// TIA Portal V19 export
TYPE "C301_VAR_IF_VEN_TYPIC"
   STRUCT
      STS_AAN { ExternalAccessible := 'False'; ExternalVisible := 'False'; ExternalWritable := 'False'} : Bool;   // TRUE = Ventilator is aangestuurd FALSE = Uit
      DIR_POS { ExternalAccessible := 'False'; ExternalVisible := 'False'; ExternalWritable := 'False'} : Bool;   // TRUE = Ventilator draait in positieve richting (rijrichting)
      DIR_NEG { ExternalAccessible := 'False'; ExternalVisible := 'False'; ExternalWritable := 'False'} : Bool;   // TRUE = Ventilator draait in negatieve richting (tegenrij)
      BMO_HAND { ExternalAccessible := 'False'; ExternalVisible := 'False'; ExternalWritable := 'False'} : Bool;   // TRUE = Ventilator in hand geschakeld FALSE = niet in hand
      TYD_TOT_AAN { ExternalAccessible := 'False'; ExternalVisible := 'False'; ExternalWritable := 'False'} : LInt;   // Totaal aantal draaiuren
      TYD_TOT_AAN_UUR { ExternalAccessible := 'False'; ExternalVisible := 'False'; ExternalWritable := 'False'} : LInt;   // Totaal aantal draaiuren
      ENE_MWA1 { ExternalAccessible := 'False'; ExternalVisible := 'False'; ExternalWritable := 'False'} : Real;   // Stroommeting fase 1
      ENE_MWA2 { ExternalAccessible := 'False'; ExternalVisible := 'False'; ExternalWritable := 'False'} : Real;   // Stroommeting fase 2
      ENE_MWA3 { ExternalAccessible := 'False'; ExternalVisible := 'False'; ExternalWritable := 'False'} : Real;   // Stroommeting fase 3
      TRL_MWA { ExternalAccessible := 'False'; ExternalVisible := 'False'; ExternalWritable := 'False'} : Real;   // Trillingsmeting
      EXT_AUT { ExternalAccessible := 'False'; ExternalVisible := 'False'; ExternalWritable := 'False'} : Bool;   // Externe (hoofd) beveiliging aangesproken
      EXT_HW { ExternalAccessible := 'False'; ExternalVisible := 'False'; ExternalWritable := 'False'} : Bool;   // Sturings hardware (PLC) in storing
      STO { ExternalAccessible := 'False'; ExternalVisible := 'False'; ExternalWritable := 'False'} : Struct   // Opsomming van alle storingen en meldingen
         A001 : Bool;   // Beveiliging aangesproken
         A002 : Bool;   // Algemene storing MCC
         A003 : Bool;   // Te hoge temperatuur in de wikkelingen van de motor van de ventilator
         A004 : Bool;   // De ventilator is in onbalans
         A005 : Bool;   // Fout stroommeting fase 1
         A006 : Bool;   // Fout stroommeting fase 2
         A007 : Bool;   // Fout stroommeting fase 3
         A008 : Bool;   // Motorlade uitgeschakeld
         A009 : Bool;   // Motorlade in test
         A010 : Bool;   // Motorlade uitgereden
         A011 : Bool;   // Draadbreuk trillingsmeting
         A012 : Bool;   // Meetbereik trillingsmeting overschreden
         AT01 : Bool;   // Discordantie motor: terugmelding niet ontvangen
         AT02 : Bool;   // Discordantie motor: terugmelding blijft aanwezig
         AT03 : Bool;   // Discordantie motor: terugmeldingen Positief en negatief tegelijkertijd
         M001 : Bool;   // Werkschakelaar uitgeschakeld
      END_STRUCT;
   END_STRUCT;
END_TYPE
